KUKA KRL program: PRUEBA02.src, PRUEBA02.dat

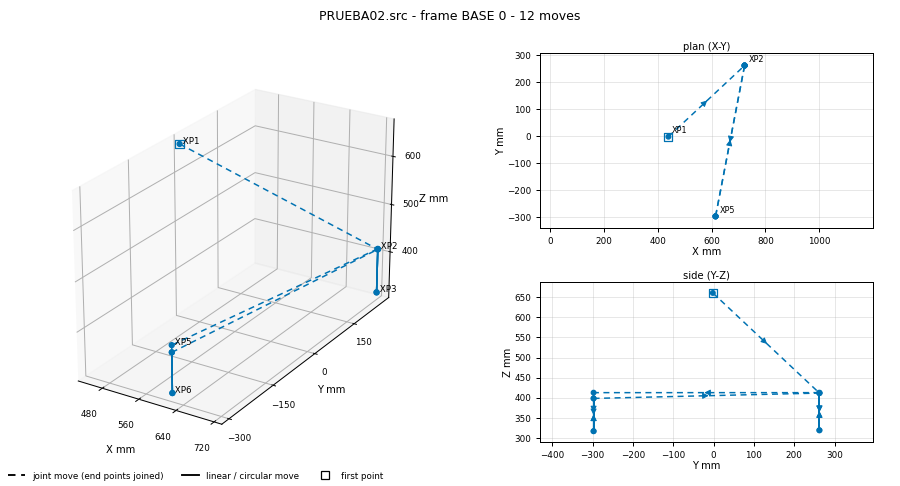
[picture p0: tool path of PRUEBA02.src in frame BASE 0, 12 of 14 moves have a stored position in this frame; points joined in program order, loops and branches not executed]
--- PRUEBA02.src ---
&ACCESS RVP
&REL 25
&PARAM EDITMASK = *
&PARAM TEMPLATE = C:\KRC\Roboter\Template\vorgabe
&PARAM DISKPATH = KRC:\R1\Program\AJEDREZ
DEF PRUEBA02( )
;FOLD INI;%{PE}
  ;FOLD BASISTECH INI
    GLOBAL INTERRUPT DECL 3 WHEN $STOPMESS==TRUE DO IR_STOPM ( )
    INTERRUPT ON 3
    BAS (#INITMOV,0 )
  ;ENDFOLD (BASISTECH INI)
  ;FOLD USER INI
    ;Make your modifications here

  ;ENDFOLD (USER INI)
;ENDFOLD (INI)

;FOLD SPTP HOME Vel=100 % DEFAULT ;%{PE}
;FOLD Parameters ;%{h}
;Params IlfProvider=kukaroboter.basistech.inlineforms.movement.spline; Kuka.IsGlobalPoint=False; Kuka.PointName=HOME; Kuka.BlendingEnabled=False; Kuka.MoveDataPtpName=DEFAULT; Kuka.VelocityPtp=100; Kuka.VelocityFieldEnabled=True; Kuka.CurrentCDSetIndex=0; Kuka.MovementParameterFieldEnabled=True; IlfCommand=SPTP
;ENDFOLD
SPTP XHOME WITH $VEL_AXIS[1] = SVEL_JOINT(100.0), $TOOL = STOOL2(FHOME), $BASE = SBASE(FHOME.BASE_NO), $IPO_MODE = SIPO_MODE(FHOME.IPO_FRAME), $LOAD = SLOAD(FHOME.TOOL_NO), $ACC_AXIS[1] = SACC_JOINT(PDEFAULT), $APO = SAPO_PTP(PDEFAULT), $GEAR_JERK[1] = SGEAR_JERK(PDEFAULT), $COLLMON_TOL_PRO[1] = USE_CM_PRO_VALUES(0)
;ENDFOLD
;FOLD Gripper SET [1]Gripper1 State=[1]ABIERTA Wait 0.2[s] Check with Strategy 1 ;%{PE}
;FOLD Parameters Parameters ;%{h}
;Params IlfProvider=GripperTech.GripperSet;setgripper=1;setstate=1;setcont=nocont;waittime=0.2;errorstrategy=1
;ENDFOLD
GRPg_SetStateAndCheck(1, 1, 0.2, 1)
;ENDFOLD

;FOLD SPTP P1 Vel=100 % PDAT1 Tool[1]:SMC Base[0] ;%{PE}
;FOLD Parameters ;%{h}
;Params IlfProvider=kukaroboter.basistech.inlineforms.movement.spline; Kuka.IsGlobalPoint=False; Kuka.PointName=P1; Kuka.BlendingEnabled=False; Kuka.MoveDataPtpName=PDAT1; Kuka.VelocityPtp=100; Kuka.VelocityFieldEnabled=True; Kuka.ColDetectFieldEnabled=True; Kuka.CurrentCDSetIndex=0; Kuka.MovementParameterFieldEnabled=True; IlfCommand=SPTP
;ENDFOLD
SPTP XP1 WITH $VEL_AXIS[1] = SVEL_JOINT(100.0), $TOOL = STOOL2(FP1), $BASE = SBASE(FP1.BASE_NO), $IPO_MODE = SIPO_MODE(FP1.IPO_FRAME), $LOAD = SLOAD(FP1.TOOL_NO), $ACC_AXIS[1] = SACC_JOINT(PPDAT1), $APO = SAPO_PTP(PPDAT1), $GEAR_JERK[1] = SGEAR_JERK(PPDAT1), $COLLMON_TOL_PRO[1] = USE_CM_PRO_VALUES(0)
;ENDFOLD
LOOP
;FOLD SPTP P2 Vel=100 % PDAT2 Tool[1]:SMC Base[0] ;%{PE}
;FOLD Parameters ;%{h}
;Params IlfProvider=kukaroboter.basistech.inlineforms.movement.spline; Kuka.IsGlobalPoint=False; Kuka.PointName=P2; Kuka.BlendingEnabled=False; Kuka.MoveDataPtpName=PDAT2; Kuka.VelocityPtp=100; Kuka.VelocityFieldEnabled=True; Kuka.ColDetectFieldEnabled=True; Kuka.CurrentCDSetIndex=0; Kuka.MovementParameterFieldEnabled=True; IlfCommand=SPTP
;ENDFOLD
SPTP XP2 WITH $VEL_AXIS[1] = SVEL_JOINT(100.0), $TOOL = STOOL2(FP2), $BASE = SBASE(FP2.BASE_NO), $IPO_MODE = SIPO_MODE(FP2.IPO_FRAME), $LOAD = SLOAD(FP2.TOOL_NO), $ACC_AXIS[1] = SACC_JOINT(PPDAT2), $APO = SAPO_PTP(PPDAT2), $GEAR_JERK[1] = SGEAR_JERK(PPDAT2), $COLLMON_TOL_PRO[1] = USE_CM_PRO_VALUES(0)
;ENDFOLD
;FOLD WAIT FOR ( IN 1 '' );%{PE}%R 8.5.19,%MKUKATPBASIS,%CEXT_WAIT_FOR,%VEXT_WAIT_FOR,%P 2:, 4:, 5:$IN, 6:1, 7:, 9:
WAIT FOR  ( $IN[1] )
;ENDFOLD
;FOLD SLIN P3 Vel=0.5 m/s CPDAT1 Tool[1]:SMC Base[0] ;%{PE}
;FOLD Parameters ;%{h}
;Params IlfProvider=kukaroboter.basistech.inlineforms.movement.spline; Kuka.IsGlobalPoint=False; Kuka.PointName=P3; Kuka.BlendingEnabled=False; Kuka.MoveDataName=CPDAT1; Kuka.VelocityPath=0.5; Kuka.VelocityFieldEnabled=True; Kuka.ColDetectFieldEnabled=True; Kuka.CurrentCDSetIndex=0; Kuka.MovementParameterFieldEnabled=True; IlfCommand=SLIN
;ENDFOLD
SLIN XP3 WITH $VEL = SVEL_CP(0.5, , LCPDAT1), $TOOL = STOOL2(FP3), $BASE = SBASE(FP3.BASE_NO), $IPO_MODE = SIPO_MODE(FP3.IPO_FRAME), $LOAD = SLOAD(FP3.TOOL_NO), $ACC = SACC_CP(LCPDAT1), $ORI_TYPE = SORI_TYP(LCPDAT1), $APO = SAPO(LCPDAT1), $JERK = SJERK(LCPDAT1), $COLLMON_TOL_PRO[1] = USE_CM_PRO_VALUES(0)
;ENDFOLD
;FOLD Gripper SET [1]Gripper1 State=[2]CERRADA Wait 0.2[s] Check with Strategy 1 ;%{PE}
;FOLD Parameters Parameters ;%{h}
;Params IlfProvider=GripperTech.GripperSet;setgripper=1;setstate=2;setcont=nocont;waittime=0.2;errorstrategy=1
;ENDFOLD
GRPg_SetStateAndCheck(1, 2, 0.2, 1)
;ENDFOLD
;FOLD SLIN P4 Vel=0.5 m/s CPDAT2 Tool[1]:SMC Base[0] ;%{PE}
;FOLD Parameters ;%{h}
;Params IlfProvider=kukaroboter.basistech.inlineforms.movement.spline; Kuka.IsGlobalPoint=False; Kuka.PointName=P4; Kuka.BlendingEnabled=False; Kuka.MoveDataName=CPDAT2; Kuka.VelocityPath=0.5; Kuka.VelocityFieldEnabled=True; Kuka.ColDetectFieldEnabled=True; Kuka.CurrentCDSetIndex=0; Kuka.MovementParameterFieldEnabled=True; IlfCommand=SLIN
;ENDFOLD
SLIN XP4 WITH $VEL = SVEL_CP(0.5, , LCPDAT2), $TOOL = STOOL2(FP4), $BASE = SBASE(FP4.BASE_NO), $IPO_MODE = SIPO_MODE(FP4.IPO_FRAME), $LOAD = SLOAD(FP4.TOOL_NO), $ACC = SACC_CP(LCPDAT2), $ORI_TYPE = SORI_TYP(LCPDAT2), $APO = SAPO(LCPDAT2), $JERK = SJERK(LCPDAT2), $COLLMON_TOL_PRO[1] = USE_CM_PRO_VALUES(0)
;ENDFOLD
;FOLD SPTP P5 Vel=100 % PDAT3 Tool[1]:SMC Base[0] ;%{PE}
;FOLD Parameters ;%{h}
;Params IlfProvider=kukaroboter.basistech.inlineforms.movement.spline; Kuka.IsGlobalPoint=False; Kuka.PointName=P5; Kuka.BlendingEnabled=False; Kuka.MoveDataPtpName=PDAT3; Kuka.VelocityPtp=100; Kuka.VelocityFieldEnabled=True; Kuka.ColDetectFieldEnabled=True; Kuka.CurrentCDSetIndex=0; Kuka.MovementParameterFieldEnabled=True; IlfCommand=SPTP
;ENDFOLD
SPTP XP5 WITH $VEL_AXIS[1] = SVEL_JOINT(100.0), $TOOL = STOOL2(FP5), $BASE = SBASE(FP5.BASE_NO), $IPO_MODE = SIPO_MODE(FP5.IPO_FRAME), $LOAD = SLOAD(FP5.TOOL_NO), $ACC_AXIS[1] = SACC_JOINT(PPDAT3), $APO = SAPO_PTP(PPDAT3), $GEAR_JERK[1] = SGEAR_JERK(PPDAT3), $COLLMON_TOL_PRO[1] = USE_CM_PRO_VALUES(0)
;ENDFOLD
;FOLD SLIN P6 Vel=0.5 m/s CPDAT3 Tool[1]:SMC Base[0] ;%{PE}
;FOLD Parameters ;%{h}
;Params IlfProvider=kukaroboter.basistech.inlineforms.movement.spline; Kuka.IsGlobalPoint=False; Kuka.PointName=P6; Kuka.BlendingEnabled=False; Kuka.MoveDataName=CPDAT3; Kuka.VelocityPath=0.5; Kuka.VelocityFieldEnabled=True; Kuka.ColDetectFieldEnabled=True; Kuka.CurrentCDSetIndex=0; Kuka.MovementParameterFieldEnabled=True; IlfCommand=SLIN
;ENDFOLD
SLIN XP6 WITH $VEL = SVEL_CP(0.5, , LCPDAT3), $TOOL = STOOL2(FP6), $BASE = SBASE(FP6.BASE_NO), $IPO_MODE = SIPO_MODE(FP6.IPO_FRAME), $LOAD = SLOAD(FP6.TOOL_NO), $ACC = SACC_CP(LCPDAT3), $ORI_TYPE = SORI_TYP(LCPDAT3), $APO = SAPO(LCPDAT3), $JERK = SJERK(LCPDAT3), $COLLMON_TOL_PRO[1] = USE_CM_PRO_VALUES(0)
;ENDFOLD
;FOLD Gripper SET [1]Gripper1 State=[1]ABIERTA Wait 0.2[s] Check with Strategy 1 ;%{PE}
;FOLD Parameters Parameters ;%{h}
;Params IlfProvider=GripperTech.GripperSet;setgripper=1;setstate=1;setcont=nocont;waittime=0.2;errorstrategy=1
;ENDFOLD
GRPg_SetStateAndCheck(1, 1, 0.2, 1)
;ENDFOLD
;FOLD SLIN P7 Vel=0.5 m/s CPDAT4 Tool[1]:SMC Base[0] ;%{PE}
;FOLD Parameters ;%{h}
;Params IlfProvider=kukaroboter.basistech.inlineforms.movement.spline; Kuka.IsGlobalPoint=False; Kuka.PointName=P7; Kuka.BlendingEnabled=False; Kuka.MoveDataName=CPDAT4; Kuka.VelocityPath=0.5; Kuka.VelocityFieldEnabled=True; Kuka.ColDetectFieldEnabled=True; Kuka.CurrentCDSetIndex=0; Kuka.MovementParameterFieldEnabled=True; IlfCommand=SLIN
;ENDFOLD
SLIN XP7 WITH $VEL = SVEL_CP(0.5, , LCPDAT4), $TOOL = STOOL2(FP7), $BASE = SBASE(FP7.BASE_NO), $IPO_MODE = SIPO_MODE(FP7.IPO_FRAME), $LOAD = SLOAD(FP7.TOOL_NO), $ACC = SACC_CP(LCPDAT4), $ORI_TYPE = SORI_TYP(LCPDAT4), $APO = SAPO(LCPDAT4), $JERK = SJERK(LCPDAT4), $COLLMON_TOL_PRO[1] = USE_CM_PRO_VALUES(0)
;ENDFOLD
;FOLD WAIT Time=5 sec;%{PE}%R 8.5.19,%MKUKATPBASIS,%CWAIT,%VWAIT,%P 3:5
WAIT SEC 5
;ENDFOLD
;FOLD SLIN P8 Vel=0.5 m/s CPDAT5 Tool[1]:SMC Base[0] ;%{PE}
;FOLD Parameters ;%{h}
;Params IlfProvider=kukaroboter.basistech.inlineforms.movement.spline; Kuka.IsGlobalPoint=False; Kuka.PointName=P8; Kuka.BlendingEnabled=False; Kuka.MoveDataName=CPDAT5; Kuka.VelocityPath=0.5; Kuka.VelocityFieldEnabled=True; Kuka.ColDetectFieldEnabled=True; Kuka.CurrentCDSetIndex=0; Kuka.MovementParameterFieldEnabled=True; IlfCommand=SLIN
;ENDFOLD
SLIN XP8 WITH $VEL = SVEL_CP(0.5, , LCPDAT5), $TOOL = STOOL2(FP8), $BASE = SBASE(FP8.BASE_NO), $IPO_MODE = SIPO_MODE(FP8.IPO_FRAME), $LOAD = SLOAD(FP8.TOOL_NO), $ACC = SACC_CP(LCPDAT5), $ORI_TYPE = SORI_TYP(LCPDAT5), $APO = SAPO(LCPDAT5), $JERK = SJERK(LCPDAT5), $COLLMON_TOL_PRO[1] = USE_CM_PRO_VALUES(0)
;ENDFOLD
;FOLD Gripper SET [1]Gripper1 State=[2]CERRADA Wait 0.2[s] Check with Strategy 1 ;%{PE}
;FOLD Parameters Parameters ;%{h}
;Params IlfProvider=GripperTech.GripperSet;setgripper=1;setstate=2;setcont=nocont;waittime=0.2;errorstrategy=1
;ENDFOLD
GRPg_SetStateAndCheck(1, 2, 0.2, 1)
;ENDFOLD
;FOLD SLIN P9 Vel=0.5 m/s CPDAT6 Tool[1]:SMC Base[0] ;%{PE}
;FOLD Parameters ;%{h}
;Params IlfProvider=kukaroboter.basistech.inlineforms.movement.spline; Kuka.IsGlobalPoint=False; Kuka.PointName=P9; Kuka.BlendingEnabled=False; Kuka.MoveDataName=CPDAT6; Kuka.VelocityPath=0.5; Kuka.VelocityFieldEnabled=True; Kuka.ColDetectFieldEnabled=True; Kuka.CurrentCDSetIndex=0; Kuka.MovementParameterFieldEnabled=True; IlfCommand=SLIN
;ENDFOLD
SLIN XP9 WITH $VEL = SVEL_CP(0.5, , LCPDAT6), $TOOL = STOOL2(FP9), $BASE = SBASE(FP9.BASE_NO), $IPO_MODE = SIPO_MODE(FP9.IPO_FRAME), $LOAD = SLOAD(FP9.TOOL_NO), $ACC = SACC_CP(LCPDAT6), $ORI_TYPE = SORI_TYP(LCPDAT6), $APO = SAPO(LCPDAT6), $JERK = SJERK(LCPDAT6), $COLLMON_TOL_PRO[1] = USE_CM_PRO_VALUES(0)
;ENDFOLD
;FOLD SPTP P10 Vel=100 % PDAT4 Tool[1]:SMC Base[0] ;%{PE}
;FOLD Parameters ;%{h}
;Params IlfProvider=kukaroboter.basistech.inlineforms.movement.spline; Kuka.IsGlobalPoint=False; Kuka.PointName=P10; Kuka.BlendingEnabled=False; Kuka.MoveDataPtpName=PDAT4; Kuka.VelocityPtp=100; Kuka.VelocityFieldEnabled=True; Kuka.ColDetectFieldEnabled=True; Kuka.CurrentCDSetIndex=0; Kuka.MovementParameterFieldEnabled=True; IlfCommand=SPTP
;ENDFOLD
SPTP XP10 WITH $VEL_AXIS[1] = SVEL_JOINT(100.0), $TOOL = STOOL2(FP10), $BASE = SBASE(FP10.BASE_NO), $IPO_MODE = SIPO_MODE(FP10.IPO_FRAME), $LOAD = SLOAD(FP10.TOOL_NO), $ACC_AXIS[1] = SACC_JOINT(PPDAT4), $APO = SAPO_PTP(PPDAT4), $GEAR_JERK[1] = SGEAR_JERK(PPDAT4), $COLLMON_TOL_PRO[1] = USE_CM_PRO_VALUES(0)
;ENDFOLD
;FOLD SLIN P11 Vel=0.5 m/s CPDAT7 Tool[1]:SMC Base[0] ;%{PE}
;FOLD Parameters ;%{h}
;Params IlfProvider=kukaroboter.basistech.inlineforms.movement.spline; Kuka.IsGlobalPoint=False; Kuka.PointName=P11; Kuka.BlendingEnabled=False; Kuka.MoveDataName=CPDAT7; Kuka.VelocityPath=0.5; Kuka.VelocityFieldEnabled=True; Kuka.ColDetectFieldEnabled=True; Kuka.CurrentCDSetIndex=0; Kuka.MovementParameterFieldEnabled=True; IlfCommand=SLIN
;ENDFOLD
SLIN XP11 WITH $VEL = SVEL_CP(0.5, , LCPDAT7), $TOOL = STOOL2(FP11), $BASE = SBASE(FP11.BASE_NO), $IPO_MODE = SIPO_MODE(FP11.IPO_FRAME), $LOAD = SLOAD(FP11.TOOL_NO), $ACC = SACC_CP(LCPDAT7), $ORI_TYPE = SORI_TYP(LCPDAT7), $APO = SAPO(LCPDAT7), $JERK = SJERK(LCPDAT7), $COLLMON_TOL_PRO[1] = USE_CM_PRO_VALUES(0)
;ENDFOLD
;FOLD Gripper SET [1]Gripper1 State=[1]ABIERTA Wait 0.2[s] Check with Strategy 1 ;%{PE}
;FOLD Parameters Parameters ;%{h}
;Params IlfProvider=GripperTech.GripperSet;setgripper=1;setstate=1;setcont=nocont;waittime=0.2;errorstrategy=1
;ENDFOLD
GRPg_SetStateAndCheck(1, 1, 0.2, 1)
;ENDFOLD
;FOLD SLIN P12 Vel=0.5 m/s CPDAT8 Tool[1]:SMC Base[0] ;%{PE}
;FOLD Parameters ;%{h}
;Params IlfProvider=kukaroboter.basistech.inlineforms.movement.spline; Kuka.IsGlobalPoint=False; Kuka.PointName=P12; Kuka.BlendingEnabled=False; Kuka.MoveDataName=CPDAT8; Kuka.VelocityPath=0.5; Kuka.VelocityFieldEnabled=True; Kuka.ColDetectFieldEnabled=True; Kuka.CurrentCDSetIndex=0; Kuka.MovementParameterFieldEnabled=True; IlfCommand=SLIN
;ENDFOLD
SLIN XP12 WITH $VEL = SVEL_CP(0.5, , LCPDAT8), $TOOL = STOOL2(FP12), $BASE = SBASE(FP12.BASE_NO), $IPO_MODE = SIPO_MODE(FP12.IPO_FRAME), $LOAD = SLOAD(FP12.TOOL_NO), $ACC = SACC_CP(LCPDAT8), $ORI_TYPE = SORI_TYP(LCPDAT8), $APO = SAPO(LCPDAT8), $JERK = SJERK(LCPDAT8), $COLLMON_TOL_PRO[1] = USE_CM_PRO_VALUES(0)
;ENDFOLD
ENDLOOP
;FOLD SPTP HOME Vel=100 % DEFAULT ;%{PE}
;FOLD Parameters ;%{h}
;Params IlfProvider=kukaroboter.basistech.inlineforms.movement.spline; Kuka.IsGlobalPoint=False; Kuka.PointName=HOME; Kuka.BlendingEnabled=False; Kuka.MoveDataPtpName=DEFAULT; Kuka.VelocityPtp=100; Kuka.VelocityFieldEnabled=True; Kuka.CurrentCDSetIndex=0; Kuka.MovementParameterFieldEnabled=True; IlfCommand=SPTP
;ENDFOLD
SPTP XHOME WITH $VEL_AXIS[1] = SVEL_JOINT(100.0), $TOOL = STOOL2(FHOME), $BASE = SBASE(FHOME.BASE_NO), $IPO_MODE = SIPO_MODE(FHOME.IPO_FRAME), $LOAD = SLOAD(FHOME.TOOL_NO), $ACC_AXIS[1] = SACC_JOINT(PDEFAULT), $APO = SAPO_PTP(PDEFAULT), $GEAR_JERK[1] = SGEAR_JERK(PDEFAULT), $COLLMON_TOL_PRO[1] = USE_CM_PRO_VALUES(0)
;ENDFOLD

END

--- PRUEBA02.dat ---
&ACCESS RVP
&REL 25
&PARAM EDITMASK = *
&PARAM TEMPLATE = C:\KRC\Roboter\Template\vorgabe
&PARAM DISKPATH = KRC:\R1\Program\AJEDREZ
DEFDAT  PRUEBA02
;FOLD EXTERNAL DECLARATIONS;%{PE}%MKUKATPBASIS,%CEXT,%VCOMMON,%P
;FOLD BASISTECH EXT;%{PE}%MKUKATPBASIS,%CEXT,%VEXT,%P
EXT  BAS (BAS_COMMAND  :IN,REAL  :IN )
DECL INT SUCCESS
;ENDFOLD (BASISTECH EXT)
;FOLD USER EXT;%{E}%MKUKATPUSER,%CEXT,%VEXT,%P
;Make your modifications here

;ENDFOLD (USER EXT)
;ENDFOLD (EXTERNAL DECLARATIONS)
DECL E6POS XP1={X 439.884644,Y -1.72222805,Z 660.311829,A 176.169434,B 89.9283,C 176.088348,S 2,T 11,E1 0.0,E2 0.0,E3 0.0,E4 0.0,E5 0.0,E6 0.0}
DECL FDAT FP1={TOOL_NO 1,BASE_NO 0,IPO_FRAME #BASE,POINT2[] " "}
DECL PDAT PPDAT1={VEL 100.000,ACC 100.000,APO_DIST 500.000,APO_MODE #CDIS,GEAR_JERK 100.000,EXAX_IGN 0}
DECL MODULEPARAM_T LAST_TP_PARAMS={PARAMS[] "Kuka.VelocityFieldEnabled=True; Kuka.ColDetectFieldEnabled=True; Kuka.MovementParameterFieldEnabled=True; Kuka.IsAngleEnabled=False; Kuka.PointName=P12; Kuka.FrameData.base_no=0; Kuka.FrameData.tool_no=1; Kuka.FrameData.ipo_frame=#BASE; Kuka.isglobalpoint=False; Kuka.MoveDataPtpName=PDAT4; Kuka.MovementDataPdat.apo_mode=#CDIS; Kuka.MovementDataPdat.apo_dist=500; Kuka.MovementData.vel=0.5; Kuka.MovementData.acc=100; Kuka.MovementData.gear_jerk=100; Kuka.MovementData.exax_ign=0; Kuka.VelocityPtp=100; Kuka.BlendingEnabled=False; Kuka.CurrentCDSetIndex=0; Kuka.MoveDataName=CPDAT8; Kuka.MovementData.apo_fac=50; Kuka.MovementData.apo_dist=500; Kuka.MovementData.axis_acc=100; Kuka.MovementData.axis_vel=100; Kuka.MovementData.circ_typ=#BASE; Kuka.MovementData.jerk_fac=50; Kuka.MovementData.ori_typ=#VAR; Kuka.VelocityPath=0.5                           "}
DECL E6POS XP2={X 722.773438,Y 262.531097,Z 412.086792,A -177.826920,B 89.9053650,C -177.909805,S 2,T 43,E1 0.0,E2 0.0,E3 0.0,E4 0.0,E5 0.0,E6 0.0}
DECL FDAT FP2={TOOL_NO 1,BASE_NO 0,IPO_FRAME #BASE,POINT2[] " "}
DECL PDAT PPDAT2={VEL 100.000,ACC 100.000,APO_DIST 500.000,APO_MODE #CDIS,GEAR_JERK 100.000,EXAX_IGN 0}
DECL E6POS XP3={X 722.773438,Y 262.531097,Z 319.826,A -177.826920,B 89.9053650,C -177.909805,S 2,T 43,E1 0.0,E2 0.0,E3 0.0,E4 0.0,E5 0.0,E6 0.0}
DECL FDAT FP3={TOOL_NO 1,BASE_NO 0,IPO_FRAME #BASE,POINT2[] " "}
DECL LDAT LCPDAT1={VEL 0.500000,ACC 100.000,APO_DIST 500.000,APO_FAC 50.0000,AXIS_VEL 100.000,AXIS_ACC 100.000,ORI_TYP #VAR,CIRC_TYP #BASE,JERK_FAC 50.0000,GEAR_JERK 100.000,EXAX_IGN 0}
DECL E6POS XP4={X 722.773438,Y 262.531097,Z 413.153809,A -177.826920,B 89.9053650,C -177.909805,S 2,T 43,E1 0.0,E2 0.0,E3 0.0,E4 0.0,E5 0.0,E6 0.0}
DECL FDAT FP4={TOOL_NO 1,BASE_NO 0,IPO_FRAME #BASE,POINT2[] " "}
DECL LDAT LCPDAT2={VEL 0.500000,ACC 100.000,APO_DIST 500.000,APO_FAC 50.0000,AXIS_VEL 100.000,AXIS_ACC 100.000,ORI_TYP #VAR,CIRC_TYP #BASE,JERK_FAC 50.0000,GEAR_JERK 100.000,EXAX_IGN 0}
DECL E6POS XP5={X 614.936340,Y -297.313385,Z 413.126404,A -177.281784,B 89.9022751,C -177.372131,S 2,T 2,E1 0.0,E2 0.0,E3 0.0,E4 0.0,E5 0.0,E6 0.0}
DECL FDAT FP5={TOOL_NO 1,BASE_NO 0,IPO_FRAME #BASE,POINT2[] " "}
DECL PDAT PPDAT3={VEL 100.000,ACC 100.000,APO_DIST 500.000,APO_MODE #CDIS,GEAR_JERK 100.000,EXAX_IGN 0}
DECL E6POS XP6={X 614.940308,Y -297.315277,Z 317.561981,A -177.103668,B 89.9028397,C -177.194031,S 2,T 2,E1 0.0,E2 0.0,E3 0.0,E4 0.0,E5 0.0,E6 0.0}
DECL FDAT FP6={TOOL_NO 1,BASE_NO 0,IPO_FRAME #BASE,POINT2[] " "}
DECL LDAT LCPDAT3={VEL 0.500000,ACC 100.000,APO_DIST 500.000,APO_FAC 50.0000,AXIS_VEL 100.000,AXIS_ACC 100.000,ORI_TYP #VAR,CIRC_TYP #BASE,JERK_FAC 50.0000,GEAR_JERK 100.000,EXAX_IGN 0}
DECL E6POS XP7={X 614.940308,Y -297.315277,Z 398.837,A -177.103683,B 89.9028397,C -177.194031,S 2,T 2,E1 0.0,E2 0.0,E3 0.0,E4 0.0,E5 0.0,E6 0.0}
DECL FDAT FP7={TOOL_NO 1,BASE_NO 0,IPO_FRAME #BASE,POINT2[] " "}
DECL LDAT LCPDAT4={VEL 0.500000,ACC 100.000,APO_DIST 500.000,APO_FAC 50.0000,AXIS_VEL 100.000,AXIS_ACC 100.000,ORI_TYP #VAR,CIRC_TYP #BASE,JERK_FAC 50.0000,GEAR_JERK 100.000,EXAX_IGN 0}
DECL E6POS XP8={X 614.940308,Y -297.315277,Z 317.561981,A -177.103668,B 89.9028397,C -177.194031,S 2,T 2,E1 0.0,E2 0.0,E3 0.0,E4 0.0,E5 0.0,E6 0.0}
DECL FDAT FP8={TOOL_NO 1,BASE_NO 0,IPO_FRAME #BASE,POINT2[] " "}
DECL LDAT LCPDAT5={VEL 0.500000,ACC 100.000,APO_DIST 500.000,APO_FAC 50.0000,AXIS_VEL 100.000,AXIS_ACC 100.000,ORI_TYP #VAR,CIRC_TYP #BASE,JERK_FAC 50.0000,GEAR_JERK 100.000,EXAX_IGN 0}
DECL E6POS XP9={X 614.940308,Y -297.315277,Z 398.837,A -177.103668,B 89.9028397,C -177.194031,S 2,T 2,E1 0.0,E2 0.0,E3 0.0,E4 0.0,E5 0.0,E6 0.0}
DECL FDAT FP9={TOOL_NO 1,BASE_NO 0,IPO_FRAME #BASE,POINT2[] " "}
DECL LDAT LCPDAT6={VEL 0.500000,ACC 100.000,APO_DIST 500.000,APO_FAC 50.0000,AXIS_VEL 100.000,AXIS_ACC 100.000,ORI_TYP #VAR,CIRC_TYP #BASE,JERK_FAC 50.0000,GEAR_JERK 100.000,EXAX_IGN 0}
DECL E6POS XP10={X 722.773438,Y 262.531097,Z 412.086792,A -177.826920,B 89.9053650,C -177.909805,S 2,T 43,E1 0.0,E2 0.0,E3 0.0,E4 0.0,E5 0.0,E6 0.0}
DECL FDAT FP10={TOOL_NO 1,BASE_NO 0,IPO_FRAME #BASE,POINT2[] " "}
DECL PDAT PPDAT4={VEL 100.000,ACC 100.000,APO_DIST 500.000,APO_MODE #CDIS,GEAR_JERK 100.000,EXAX_IGN 0}
DECL E6POS XP11={X 722.773438,Y 262.531097,Z 319.826,A -177.826920,B 89.9053650,C -177.909805,S 2,T 43,E1 0.0,E2 0.0,E3 0.0,E4 0.0,E5 0.0,E6 0.0}
DECL FDAT FP11={TOOL_NO 1,BASE_NO 0,IPO_FRAME #BASE,POINT2[] " "}
DECL LDAT LCPDAT7={VEL 0.500000,ACC 100.000,APO_DIST 500.000,APO_FAC 50.0000,AXIS_VEL 100.000,AXIS_ACC 100.000,ORI_TYP #VAR,CIRC_TYP #BASE,JERK_FAC 50.0000,GEAR_JERK 100.000,EXAX_IGN 0}
DECL E6POS XP12={X 722.773438,Y 262.531097,Z 412.086792,A -177.826920,B 89.9053650,C -177.909805,S 2,T 43,E1 0.0,E2 0.0,E3 0.0,E4 0.0,E5 0.0,E6 0.0}
DECL FDAT FP12={TOOL_NO 1,BASE_NO 0,IPO_FRAME #BASE,POINT2[] " "}
DECL LDAT LCPDAT8={VEL 0.500000,ACC 100.000,APO_DIST 500.000,APO_FAC 50.0000,AXIS_VEL 100.000,AXIS_ACC 100.000,ORI_TYP #VAR,CIRC_TYP #BASE,JERK_FAC 50.0000,GEAR_JERK 100.000,EXAX_IGN 0}
ENDDAT
